PROGRAM PRG_TEST_FB_PARLOGGING
VAR
	fbParLogging 	: FB_ParameterFileHandler;
	//fbParLogging 	: Fb_ParLogging;
	stParameter 	: Udt_Parameter; // NOTE: Udt_Parameter is persistent
	bAddParameter 	: BOOL;
	bInit			: BOOL;
END_VAR

fbParLogging();

IF bAddParameter THEN
	bAddParameter := FALSE;
	fbParLogging.CmdAddParameter(stParameter);
END_IF

IF bInit THEN
	bInit R= fbParLogging.Init();
END_IF

END_PROGRAM

(* stored: Version 1.1.0.1, ProductVersion 3.1.4024.11
   POU PRG_TEST_FB_PARLOGGING: Id {9f293204-c2aa-0fe1-1474-f57aeffff999}, SpecialFunc None *)
